(* CODESYS project sixaxis.project

Project tree, tasks and I/O mapping:
  Device : CODESYS Control Win V3, 3S - Smart Software Solutions GmbH, version 3.5.17.0
    application Application
      libraries: VisuDialogs, * (System)
      task VISU_TASK (cyclic, interval 100 ms, priority 10) calls VisuElems.Visu_Prg
      task Task (cyclic, interval t#4ms, priority 1) calls PowerNCam
      visualisation Visualization
      visualisation Visualization_1
      CAM/
        Cam1
        Cam2
        Cam3
        CamA
        CamB
        CamC
        CamD
        CamE
      Motion/
        program PowerNCam [FBD]
    SoftMotion General Axis Pool : SoftMotion General Axis Pool, 3S - Smart Software Solutions GmbH, version 4.11.0.0
      Serv1 : SM_Drive_Virtual, 3S - Smart Software Solutions GmbH, order no. 1805, version 4.0.0.0
          settings: wDriveID = 0; iMovementType = 0; fSWMaxVelocity = 1e3; fSWMaxAcceleration = 1e5; fSWMaxDeceleration = 1e5; fRampJerk = 1e7; fSWLimitPositive = 100.0
      Master : SM_Drive_Virtual, 3S - Smart Software Solutions GmbH, order no. 1805, version 4.0.0.0
          settings: iMovementType = 0; fPositionPeriod = 360; fSWMaxVelocity = 1e3; fSWMaxAcceleration = 1e5; fSWMaxDeceleration = 1e5; fRampJerk = 1e7
      Serv2 : SM_Drive_Virtual, 3S - Smart Software Solutions GmbH, order no. 1805, version 4.0.0.0
          settings: wDriveID = 2; iMovementType = 0; fSWMaxVelocity = 1e3; fSWMaxAcceleration = 1e5; fSWMaxDeceleration = 1e5
      Serv3 : SM_Drive_Virtual, 3S - Smart Software Solutions GmbH, order no. 1805, version 4.0.0.0
          settings: wDriveID = 3; iMovementType = 0
      Serv4 : SM_Drive_Virtual, 3S - Smart Software Solutions GmbH, order no. 1805, version 4.0.0.0
          settings: wDriveID = 4; iMovementType = 0
      Serv5 : SM_Drive_Virtual, 3S - Smart Software Solutions GmbH, order no. 1805, version 4.0.0.0
          settings: wDriveID = 5; iMovementType = 0
  libraries: Standard, 3.5.18.0 (System)
  text list GlobalTextList
  GlobalImagePool
*)

// Device/Application/Motion/PowerNCam
PROGRAM PowerNCam
VAR
	power1,power2,power3,power4,power5,power6: MC_Power;
	SanalMaster: MC_MoveVelocity;
	EXE: BOOL;
	SETLE:BOOL;
	
	Secim1,Secim2,Secim3,Secim4,Secim5: MC_CamTableSelect;
	Camyaz1,Camyaz2,Camyaz3,Camyaz4,Camyaz5: MC_CamIn;
	Camset1,Camset2,Camset3,Camset4,Camset5: SMC_GetCamSlaveSetPosition;
	
	//CAM1<<
	Eks1: ARRAY[0..3] OF SMC_CAMXYVA := [
        (dX := 0, dY := 0, dV := 0, dA := 0),
        (dX := 120, dY := 100, dV := 0, dA := 0),
        (dX := 240, dY := 300, dV := 0, dA := 0),
        (dX := 360, dY := 360, dV := 0, dA := 0)];
		//Ust kisimdaki degerler yerine degisken atayarak
		//cam tablosunu makine calisir iken guncelleyebiliriz.
	CamA: MC_CAM_REF := (nElements := 4, byType := 3, xStart := 0, 
	xEnd := 360, nTappets := 0, strCAMName := 'Eks1', 
	pce := ADR(Eks1), xPartofLM := TRUE);
	
	Eks2: ARRAY[0..3] OF SMC_CAMXYVA := [
        (dX := 0, dY := 0, dV := 0, dA := 0),
        (dX := 120, dY := 100, dV := 0, dA := 0),
        (dX := 240, dY := 300, dV := 0, dA := 0),
        (dX := 360, dY := 360, dV := 0, dA := 0)];
		//Ust kisimdaki degerler yerine degisken atayarak
		//cam tablosunu makine calisir iken guncelleyebiliriz.
	CamB: MC_CAM_REF := (nElements := 4, byType := 3, xStart := 0, 
	xEnd := 360, nTappets := 0, strCAMName := 'Eks2', 
	pce := ADR(Eks2), xPartofLM := TRUE);
	
	Eks3: ARRAY[0..3] OF SMC_CAMXYVA := [
        (dX := 0, dY := 0, dV := 0, dA := 0),
        (dX := 120, dY := 100, dV := 0, dA := 0),
        (dX := 240, dY := 300, dV := 0, dA := 0),
        (dX := 360, dY := 360, dV := 0, dA := 0)];
		//Ust kisimdaki degerler yerine degisken atayarak
		//cam tablosunu makine calisir iken guncelleyebiliriz.
	CamC: MC_CAM_REF := (nElements := 4, byType := 3, xStart := 0, 
	xEnd := 360, nTappets := 0, strCAMName := 'Eks3', 
	pce := ADR(Eks3), xPartofLM := TRUE);
	
	Eks4: ARRAY[0..3] OF SMC_CAMXYVA := [
        (dX := 0, dY := 0, dV := 0, dA := 0),
        (dX := 120, dY := 100, dV := 0, dA := 0),
        (dX := 240, dY := 300, dV := 0, dA := 0),
        (dX := 360, dY := 360, dV := 0, dA := 0)];
		//Ust kisimdaki degerler yerine degisken atayarak
		//cam tablosunu makine calisir iken guncelleyebiliriz.
	CamD: MC_CAM_REF := (nElements := 4, byType := 3, xStart := 0, 
	xEnd := 360, nTappets := 0, strCAMName := 'Eks4', 
	pce := ADR(Eks4), xPartofLM := TRUE);
	
	Eks5: ARRAY[0..3] OF SMC_CAMXYVA := [
        (dX := 0, dY := 0, dV := 0, dA := 0),
        (dX := 120, dY := 100, dV := 0, dA := 0),
        (dX := 240, dY := 300, dV := 0, dA := 0),
        (dX := 360, dY := 360, dV := 0, dA := 0)];
		//Ust kisimdaki degerler yerine degisken atayarak
		//cam tablosunu makine calisir iken guncelleyebiliriz.
	CamE: MC_CAM_REF := (nElements := 4, byType := 3, xStart := 0, 
	xEnd := 360, nTappets := 0, strCAMName := 'Eks5', 
	pce := ADR(Eks5), xPartofLM := TRUE);
	
	SMC_CamEditor_1: SMC_CamEditor;
	SMC_CamEditor_2: SMC_CamEditor;
	SMC_CamEditor_3: SMC_CamEditor;
	SMC_CamEditor_4: SMC_CamEditor;
	SMC_CamEditor_5: SMC_CamEditor;
	Sign1: BOOL;
	Sign2: BOOL;
	Sign3: BOOL;
	Sign4: BOOL;
	MC_ReadActualPosition_0: MC_ReadActualPosition;
	SR_0: SR;
	SER: SR;
END_VAR

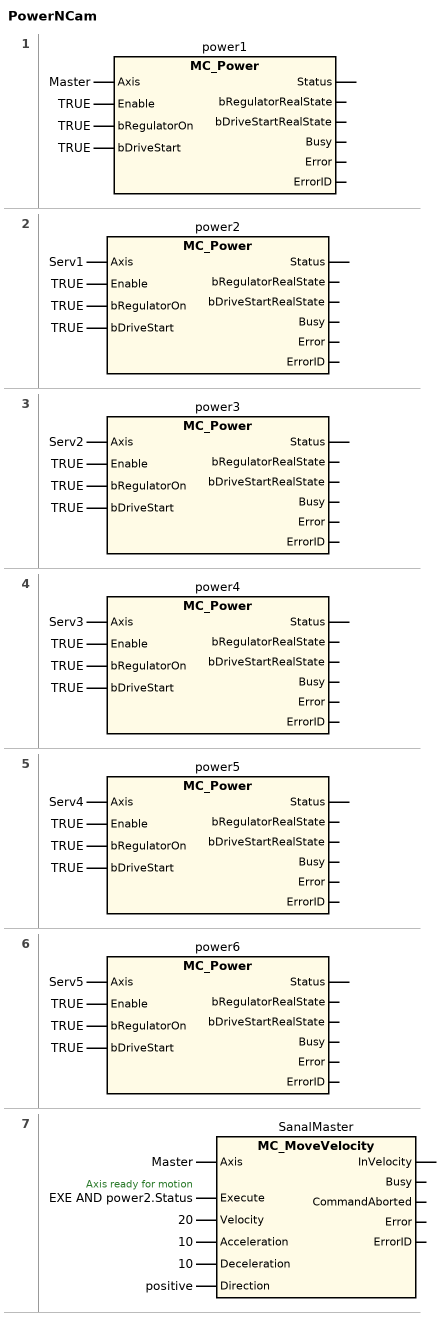
// NETWORK 1
power1(Axis := Master, Enable := TRUE, bRegulatorOn := TRUE, bDriveStart := TRUE); // MC_Power

// NETWORK 2
power2(Axis := Serv1, Enable := TRUE, bRegulatorOn := TRUE, bDriveStart := TRUE); // MC_Power

// NETWORK 3
power3(Axis := Serv2, Enable := TRUE, bRegulatorOn := TRUE, bDriveStart := TRUE); // MC_Power

// NETWORK 4
power4(Axis := Serv3, Enable := TRUE, bRegulatorOn := TRUE, bDriveStart := TRUE); // MC_Power

// NETWORK 5
power5(Axis := Serv4, Enable := TRUE, bRegulatorOn := TRUE, bDriveStart := TRUE); // MC_Power

// NETWORK 6
power6(Axis := Serv5, Enable := TRUE, bRegulatorOn := TRUE, bDriveStart := TRUE); // MC_Power

// NETWORK 7
//   EXE AND power2.Status: Axis ready for motion
SanalMaster(
    Axis := Master,
    Execute := EXE AND power2.Status,
    Velocity := 20,
    Acceleration := 10,
    Deceleration := 10,
    Direction := positive); // MC_MoveVelocity

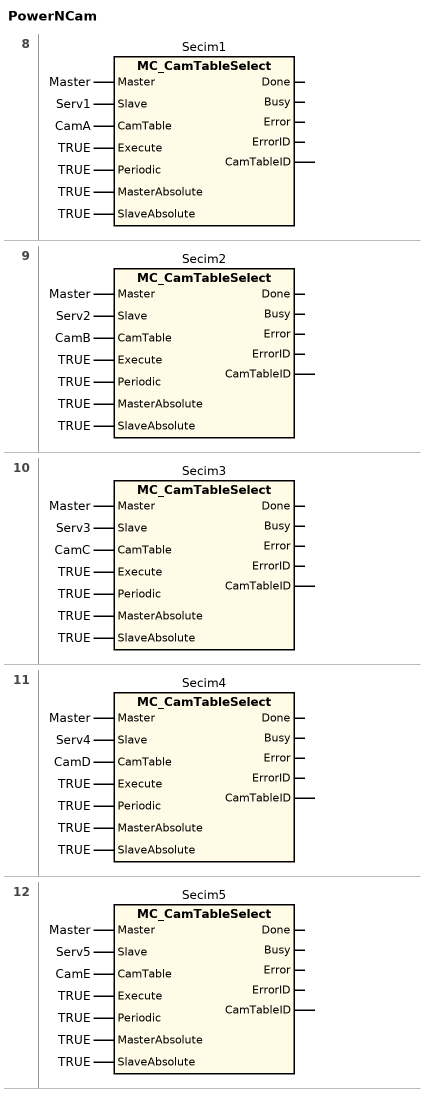
// NETWORK 8
Secim1(
    Master := Master,
    Slave := Serv1,
    CamTable := CamA,
    Execute := TRUE,
    Periodic := TRUE,
    MasterAbsolute := TRUE,
    SlaveAbsolute := TRUE); // MC_CamTableSelect

// NETWORK 9
Secim2(
    Master := Master,
    Slave := Serv2,
    CamTable := CamB,
    Execute := TRUE,
    Periodic := TRUE,
    MasterAbsolute := TRUE,
    SlaveAbsolute := TRUE); // MC_CamTableSelect

// NETWORK 10
Secim3(
    Master := Master,
    Slave := Serv3,
    CamTable := CamC,
    Execute := TRUE,
    Periodic := TRUE,
    MasterAbsolute := TRUE,
    SlaveAbsolute := TRUE); // MC_CamTableSelect

// NETWORK 11
Secim4(
    Master := Master,
    Slave := Serv4,
    CamTable := CamD,
    Execute := TRUE,
    Periodic := TRUE,
    MasterAbsolute := TRUE,
    SlaveAbsolute := TRUE); // MC_CamTableSelect

// NETWORK 12
Secim5(
    Master := Master,
    Slave := Serv5,
    CamTable := CamE,
    Execute := TRUE,
    Periodic := TRUE,
    MasterAbsolute := TRUE,
    SlaveAbsolute := TRUE); // MC_CamTableSelect

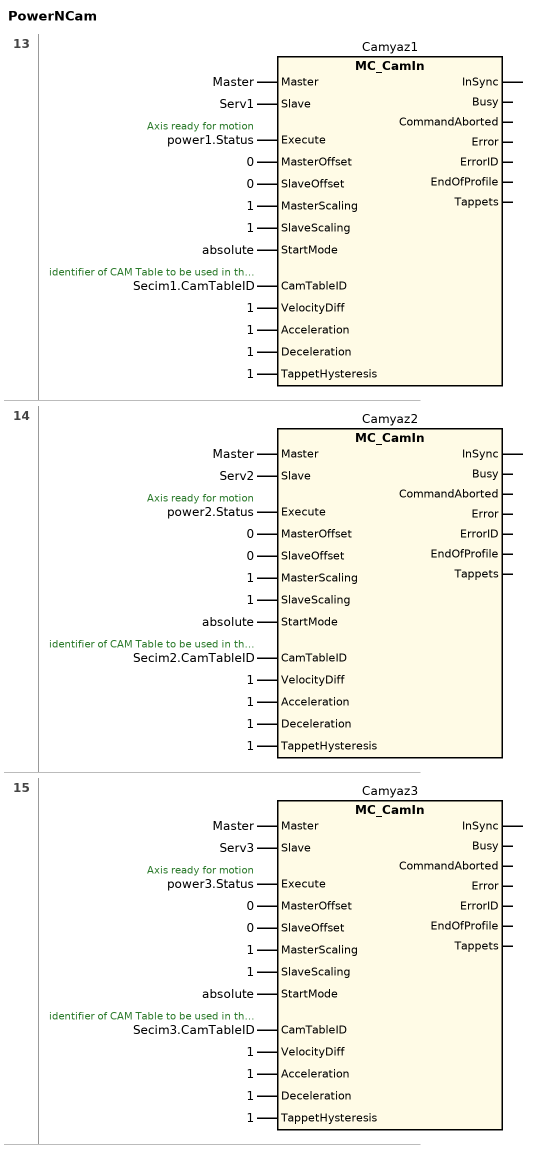
// NETWORK 13
//   power1.Status: Axis ready for motion
//   Secim1.CamTableID: identifier of CAM Table to be used in the MC_CamIn FB
Camyaz1(
    Master := Master,
    Slave := Serv1,
    Execute := power1.Status,
    MasterOffset := 0,
    SlaveOffset := 0,
    MasterScaling := 1,
    SlaveScaling := 1,
    StartMode := absolute,
    CamTableID := Secim1.CamTableID,
    VelocityDiff := 1,
    Acceleration := 1,
    Deceleration := 1,
    TappetHysteresis := 1); // MC_CamIn

// NETWORK 14
//   power2.Status: Axis ready for motion
//   Secim2.CamTableID: identifier of CAM Table to be used in the MC_CamIn FB
Camyaz2(
    Master := Master,
    Slave := Serv2,
    Execute := power2.Status,
    MasterOffset := 0,
    SlaveOffset := 0,
    MasterScaling := 1,
    SlaveScaling := 1,
    StartMode := absolute,
    CamTableID := Secim2.CamTableID,
    VelocityDiff := 1,
    Acceleration := 1,
    Deceleration := 1,
    TappetHysteresis := 1); // MC_CamIn

// NETWORK 15
//   power3.Status: Axis ready for motion
//   Secim3.CamTableID: identifier of CAM Table to be used in the MC_CamIn FB
Camyaz3(
    Master := Master,
    Slave := Serv3,
    Execute := power3.Status,
    MasterOffset := 0,
    SlaveOffset := 0,
    MasterScaling := 1,
    SlaveScaling := 1,
    StartMode := absolute,
    CamTableID := Secim3.CamTableID,
    VelocityDiff := 1,
    Acceleration := 1,
    Deceleration := 1,
    TappetHysteresis := 1); // MC_CamIn

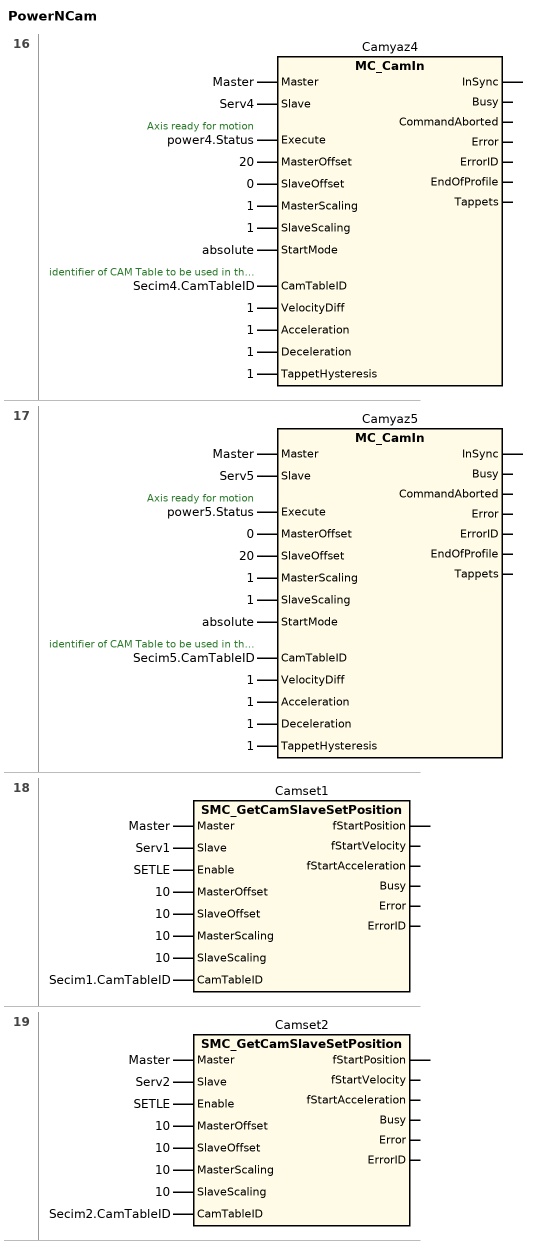
// NETWORK 16
//   power4.Status: Axis ready for motion
//   Secim4.CamTableID: identifier of CAM Table to be used in the MC_CamIn FB
Camyaz4(
    Master := Master,
    Slave := Serv4,
    Execute := power4.Status,
    MasterOffset := 20,
    SlaveOffset := 0,
    MasterScaling := 1,
    SlaveScaling := 1,
    StartMode := absolute,
    CamTableID := Secim4.CamTableID,
    VelocityDiff := 1,
    Acceleration := 1,
    Deceleration := 1,
    TappetHysteresis := 1); // MC_CamIn

// NETWORK 17
//   power5.Status: Axis ready for motion
//   Secim5.CamTableID: identifier of CAM Table to be used in the MC_CamIn FB
Camyaz5(
    Master := Master,
    Slave := Serv5,
    Execute := power5.Status,
    MasterOffset := 0,
    SlaveOffset := 20,
    MasterScaling := 1,
    SlaveScaling := 1,
    StartMode := absolute,
    CamTableID := Secim5.CamTableID,
    VelocityDiff := 1,
    Acceleration := 1,
    Deceleration := 1,
    TappetHysteresis := 1); // MC_CamIn

// NETWORK 18
Camset1(
    Master := Master,
    Slave := Serv1,
    Enable := SETLE,
    MasterOffset := 10,
    SlaveOffset := 10,
    MasterScaling := 10,
    SlaveScaling := 10,
    CamTableID := Secim1.CamTableID); // SMC_GetCamSlaveSetPosition

// NETWORK 19
Camset2(
    Master := Master,
    Slave := Serv2,
    Enable := SETLE,
    MasterOffset := 10,
    SlaveOffset := 10,
    MasterScaling := 10,
    SlaveScaling := 10,
    CamTableID := Secim2.CamTableID); // SMC_GetCamSlaveSetPosition

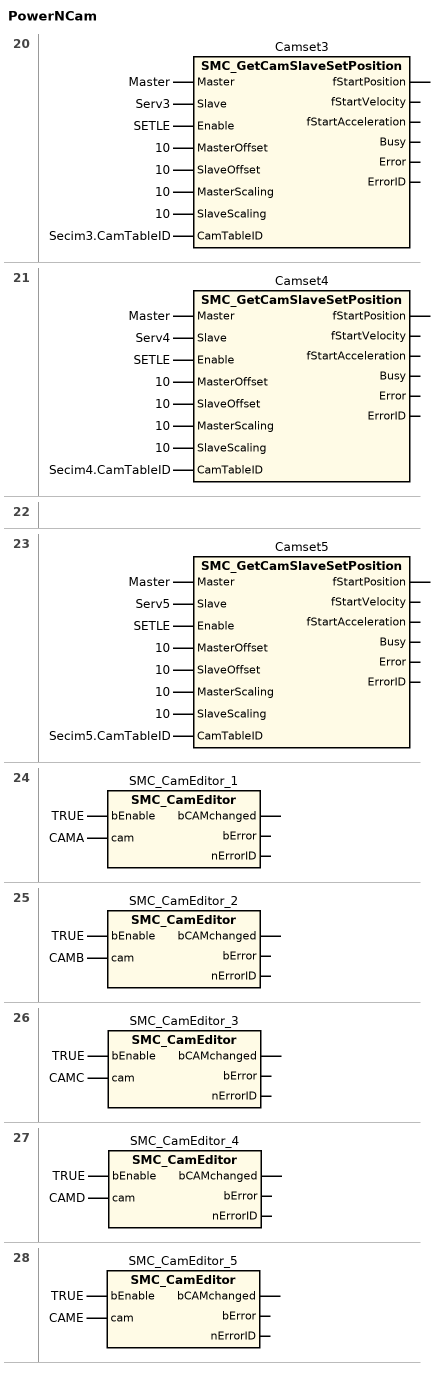
// NETWORK 20
Camset3(
    Master := Master,
    Slave := Serv3,
    Enable := SETLE,
    MasterOffset := 10,
    SlaveOffset := 10,
    MasterScaling := 10,
    SlaveScaling := 10,
    CamTableID := Secim3.CamTableID); // SMC_GetCamSlaveSetPosition

// NETWORK 21
Camset4(
    Master := Master,
    Slave := Serv4,
    Enable := SETLE,
    MasterOffset := 10,
    SlaveOffset := 10,
    MasterScaling := 10,
    SlaveScaling := 10,
    CamTableID := Secim4.CamTableID); // SMC_GetCamSlaveSetPosition

// NETWORK 22

// NETWORK 23
Camset5(
    Master := Master,
    Slave := Serv5,
    Enable := SETLE,
    MasterOffset := 10,
    SlaveOffset := 10,
    MasterScaling := 10,
    SlaveScaling := 10,
    CamTableID := Secim5.CamTableID); // SMC_GetCamSlaveSetPosition

// NETWORK 24
SMC_CamEditor_1(bEnable := TRUE, cam := CAMA); // SMC_CamEditor

// NETWORK 25
SMC_CamEditor_2(bEnable := TRUE, cam := CAMB); // SMC_CamEditor

// NETWORK 26
SMC_CamEditor_3(bEnable := TRUE, cam := CAMC); // SMC_CamEditor

// NETWORK 27
SMC_CamEditor_4(bEnable := TRUE, cam := CAMD); // SMC_CamEditor

// NETWORK 28
SMC_CamEditor_5(bEnable := TRUE, cam := CAME); // SMC_CamEditor

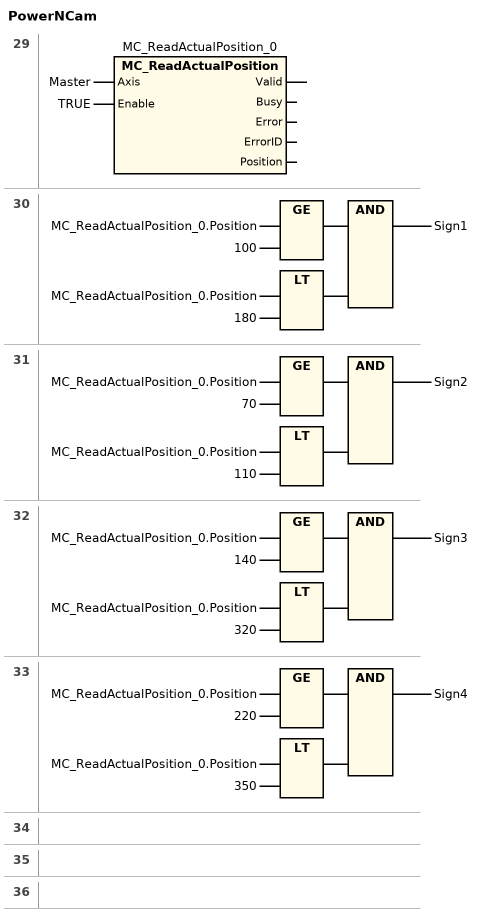
// NETWORK 29
MC_ReadActualPosition_0(Axis := Master, Enable := TRUE); // MC_ReadActualPosition

// NETWORK 30
Sign1 := MC_ReadActualPosition_0.Position >= 100 AND MC_ReadActualPosition_0.Position < 180;

// NETWORK 31
Sign2 := MC_ReadActualPosition_0.Position >= 70 AND MC_ReadActualPosition_0.Position < 110;

// NETWORK 32
Sign3 := MC_ReadActualPosition_0.Position >= 140 AND MC_ReadActualPosition_0.Position < 320;

// NETWORK 33
Sign4 := MC_ReadActualPosition_0.Position >= 220 AND MC_ReadActualPosition_0.Position < 350;

// NETWORK 34

// NETWORK 35

// NETWORK 36

END_PROGRAM

// Device/Application/Visualization
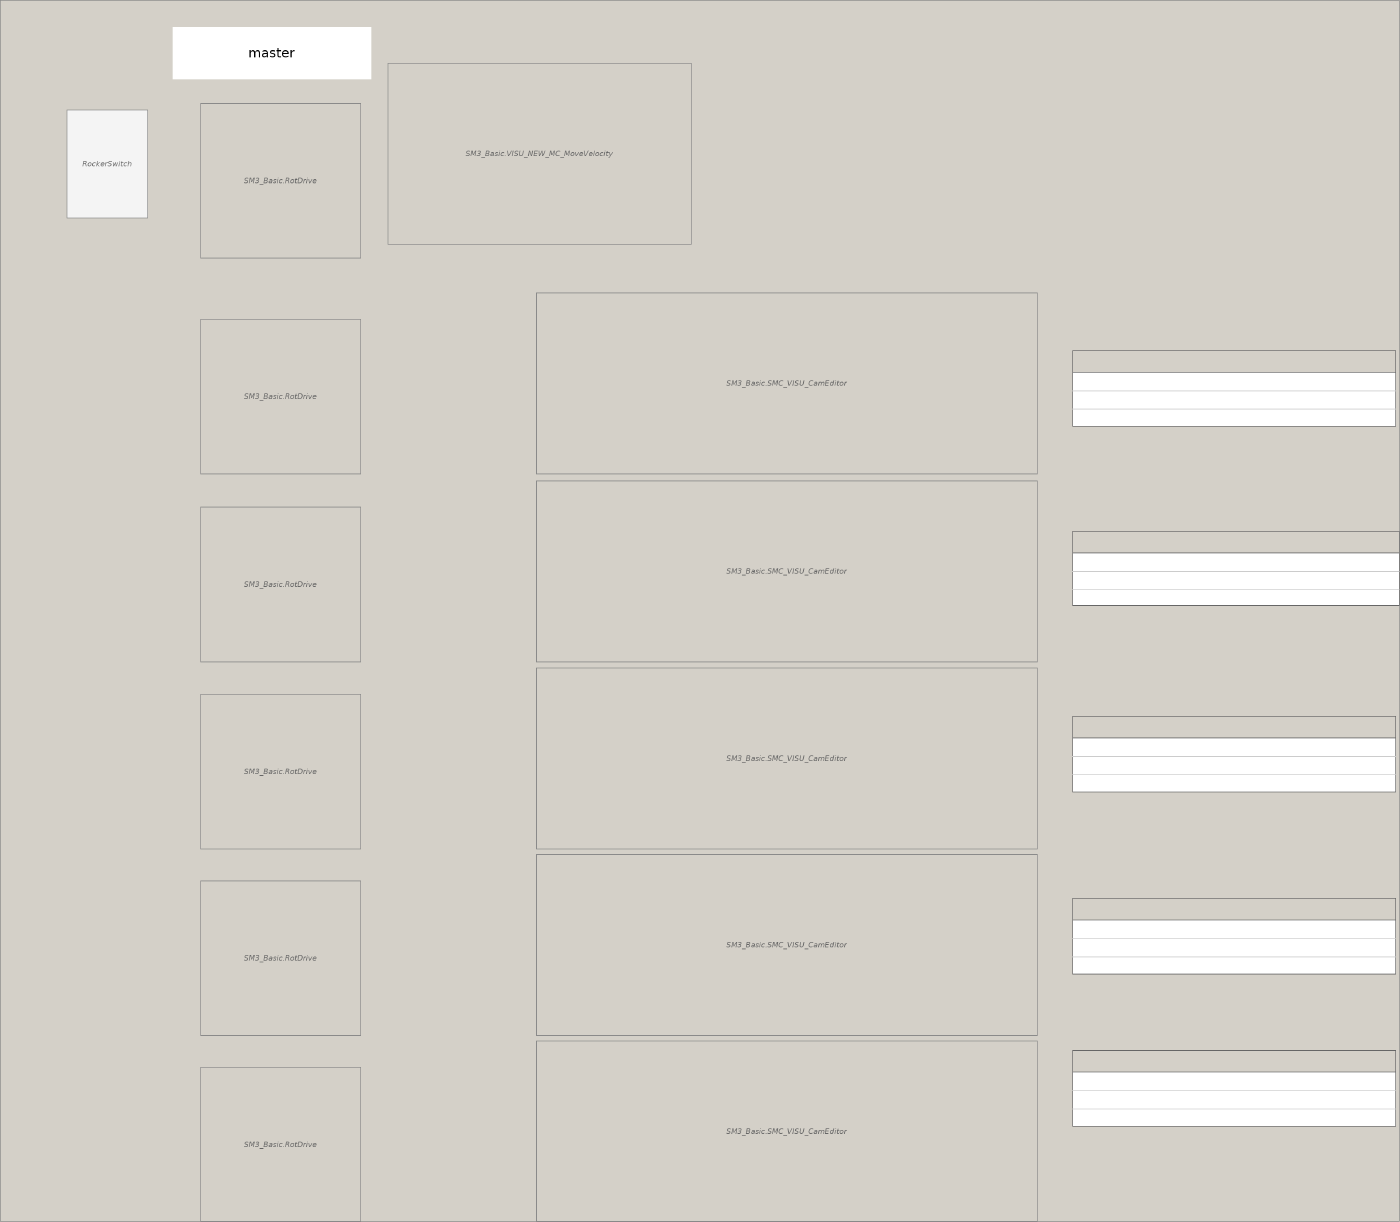
VISUALIZATION Visualization  // 1914x1671
    Frame (530,86 415x248)
        shows SM3_Basic.VISU_NEW_MC_MoveVelocity(m_Input_FB := MOTION_PRG.MoveVirtual)
    Frame (274,141 219x212)
        shows SM3_Basic.RotDrive(m_Input_AXISREF := Master)
    Frame (274,693 219x212)
        shows SM3_Basic.RotDrive(m_Input_AXISREF := IoConfig_Globals.Serv1)
    Frame (274,436 219x212)
        shows SM3_Basic.RotDrive(m_Input_AXISREF := Serv2)
    Line (74,681)
    Frame (274,949 219x212)
        shows SM3_Basic.RotDrive(m_Input_AXISREF := Serv3)
    Frame (274,1204 219x212)
        shows SM3_Basic.RotDrive(m_Input_AXISREF := Serv4)
    Frame (274,1459 219x212)
        shows SM3_Basic.RotDrive(m_Input_AXISREF := Serv5)
    Textfield (235,36 273x73), "master"
    RockerSwitch (91,150 111x148), variable: PowerNCam.EXE, behaviour: TOGGLE, style: Switch-RockerSwitch-Gray
    Frame (733,400 685x248)
        shows SM3_Basic.SMC_VISU_CamEditor(editor := PowerNCam.SMC_CamEditor_1)
    Frame (733,657 685x248)
        shows SM3_Basic.SMC_VISU_CamEditor(editor := PowerNCam.SMC_CamEditor_2)
    Frame (733,913 685x248)
        shows SM3_Basic.SMC_VISU_CamEditor(editor := PowerNCam.SMC_CamEditor_3)
    Frame (733,1168 685x248)
        shows SM3_Basic.SMC_VISU_CamEditor(editor := PowerNCam.SMC_CamEditor_4)
    Frame (733,1423 685x248)
        shows SM3_Basic.SMC_VISU_CamEditor(editor := PowerNCam.SMC_CamEditor_5)
    Table (1466,479 442x104), data array: PowerNCam.Eks1
        p1014161805: 3 - 0 + INT#1
        p3854506369: CokEksenli.Eks1[INDEX].dX
        p1892666644: CokEksenli.Eks1[INDEX].dY
        p338671338: CokEksenli.Eks1[INDEX].dV
        p2170511999: CokEksenli.Eks1[INDEX].dA
        p2232123230: Master
        p511219082: Slave
        p1755163831: Velocity
        p4092479075: Acceleration
        p2685023577: PowerNCam.Eks1[INDEX].dX
        p3312258591: PowerNCam.Eks1[INDEX].dY
        p1791247317: PowerNCam.Eks1[INDEX].dV
        p262371475: PowerNCam.Eks1[INDEX].dA
    Table (1466,726 448x102), data array: PowerNCam.Eks2
        p1014161805: 3 - 0 + INT#1
        p3854506369: CokEksenli.Eks2[INDEX].dX
        p1892666644: CokEksenli.Eks2[INDEX].dY
        p338671338: CokEksenli.Eks2[INDEX].dV
        p2170511999: CokEksenli.Eks2[INDEX].dA
        p2232123230: Master
        p511219082: Slave
        p1755163831: Velocity
        p4092479075: Acceleration
        p2685023577: PowerNCam.Eks2[INDEX].dX
        p3312258591: PowerNCam.Eks2[INDEX].dY
        p1791247317: PowerNCam.Eks2[INDEX].dV
        p262371475: PowerNCam.Eks2[INDEX].dA
    Table (1466,979 442x104), data array: PowerNCam.Eks3
        p1014161805: 3 - 0 + INT#1
        p3854506369: CokEksenli.Eks3[INDEX].dX
        p1892666644: CokEksenli.Eks3[INDEX].dY
        p338671338: CokEksenli.Eks3[INDEX].dV
        p2170511999: CokEksenli.Eks3[INDEX].dA
        p2232123230: Master
        p511219082: Slave
        p1755163831: Velocity
        p4092479075: Acceleration
        p2685023577: PowerNCam.Eks3[INDEX].dX
        p3312258591: PowerNCam.Eks3[INDEX].dY
        p1791247317: PowerNCam.Eks3[INDEX].dV
        p262371475: PowerNCam.Eks3[INDEX].dA
    Table (1466,1228 442x104), data array: PowerNCam.Eks4
        p1014161805: 3 - 0 + INT#1
        p3854506369: CokEksenli.Eks4[INDEX].dX
        p1892666644: CokEksenli.Eks4[INDEX].dY
        p338671338: CokEksenli.Eks4[INDEX].dV
        p2170511999: CokEksenli.Eks4[INDEX].dA
        p2232123230: Master
        p511219082: Slave
        p1755163831: Velocity
        p4092479075: Acceleration
        p2685023577: PowerNCam.Eks4[INDEX].dX
        p3312258591: PowerNCam.Eks4[INDEX].dY
        p1791247317: PowerNCam.Eks4[INDEX].dV
        p262371475: PowerNCam.Eks4[INDEX].dA
    Table (1466,1436 442x104), data array: PowerNCam.Eks5
        p1014161805: 3 - 0 + INT#1
        p3854506369: CokEksenli.Eks5[INDEX].dX
        p1892666644: CokEksenli.Eks5[INDEX].dY
        p338671338: CokEksenli.Eks5[INDEX].dV
        p2170511999: CokEksenli.Eks5[INDEX].dA
        p2232123230: Master
        p511219082: Slave
        p1755163831: Velocity
        p4092479075: Acceleration
        p2685023577: PowerNCam.Eks5[INDEX].dX
        p3312258591: PowerNCam.Eks5[INDEX].dY
        p1791247317: PowerNCam.Eks5[INDEX].dV
        p262371475: PowerNCam.Eks5[INDEX].dA
END_VISUALIZATION

// Device/Application/Visualization_1
VISUALIZATION Visualization_1  // 2x2
END_VISUALIZATION
